// TIA Portal V19 export
TYPE "LEXCHANGETRAY_typeSr1000ProfinetTelegram_terminalStatusBits"
// stored: Access Published
   STRUCT
      statusByte : Byte;
      in1 : Bool;
      in2 : Bool;
      out1 : Bool;
      out2 : Bool;
      out3 : Bool;
   END_STRUCT;
END_TYPE
